INTERFACE I_ListObject

METHOD PUBLIC M_Add : BOOL
VAR_INPUT
	Object: 	I_Object;
END_VAR
END_METHOD

METHOD PUBLIC M_Clear : BOOL
END_METHOD

METHOD PUBLIC M_Find : DINT
VAR_INPUT
	Object: 	I_Object;
END_VAR
END_METHOD

METHOD PUBLIC M_Index : I_Object
VAR_INPUT
	Index: 	DINT;
END_VAR
END_METHOD

METHOD PUBLIC M_Remove : BOOL
VAR_INPUT
	Object: 	I_Object;
END_VAR
END_METHOD

PROPERTY P_Length : DINT
GET
END_GET
END_PROPERTY

END_INTERFACE

(* stored: Version 1.1.0.1
   Itf I_ListObject: Id {89866f33-5c66-47f4-9f9b-486325a73916}
   Method M_Add: Id {b0452453-b851-4454-a958-0966dda80209}
   Method M_Clear: Id {71968688-9bd5-40f4-9456-85ce4eb1eae3}
   Method M_Find: Id {01e077cb-06ab-4d21-8b2c-6969a4e1dc39}
   Method M_Index: Id {dc9cac95-f4e9-4e25-9b9b-cd3acef9fb84}
   Method M_Remove: Id {e01476f8-7fdf-4b72-a251-8f25b6780dc3}
   Property P_Length: Id {8984ef33-2a6a-437c-9a3d-5db2df8c7b01}
   Get Get: Id {76fb9fa3-a119-439a-9a41-9952f355a026} *)
